FUNCTION_BLOCK ILOCK_2_E_AX (* Event-driven bistable and Toggle with Dual Interlock (Adapter) *)
  (* Standard: 61499-1 Annex A; Description: Copyright (c) 2017, 2024 fortiss GmbH, HR Agrartechnik GmbH This program and the accompanying materials are made available under the terms of the Eclipse Public License 2.0 which is available at https://www.eclipse.org/legal/epl-2.0/ SPDX-License-Identifier: EPL-2.0 *)
  (* Version 3.0, 2025-04-14, Patrick Aigner, changed package *)
  (* Version 1.1, 2024-08-27, Franz Höpfinger, HR Agrartechnik GmbH, Copy E_SR and make this FB *)
  (* Version 1.0, 2017-09-22, Alois Zoitl, fortiss GmbH, initial API and implementation and/or initial documentation *)
  PACKAGE logiBUS::signalprocessing::interlock;
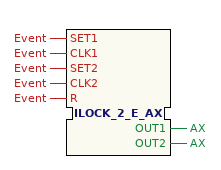
  EVENT_INPUT
    SET1; (* Set output OUT1 *)
    CLK1; (* Clock for triggering a output toggle on OUT1 *)
    SET2; (* Set output OUT2 *)
    CLK2; (* Clock for triggering a output toggle on OUT2 *)
    R; (* Reset all outputs *)
  END_EVENT
  PLUGS
    OUT1 : adapter::types::unidirectional::AX; (* value of flip flop *)
    OUT2 : adapter::types::unidirectional::AX; (* value of flip flop *)
  END_PLUGS
  VAR
    EDGE1 : BOOL := FALSE;
    EDGE2 : BOOL := FALSE;
  END_VAR
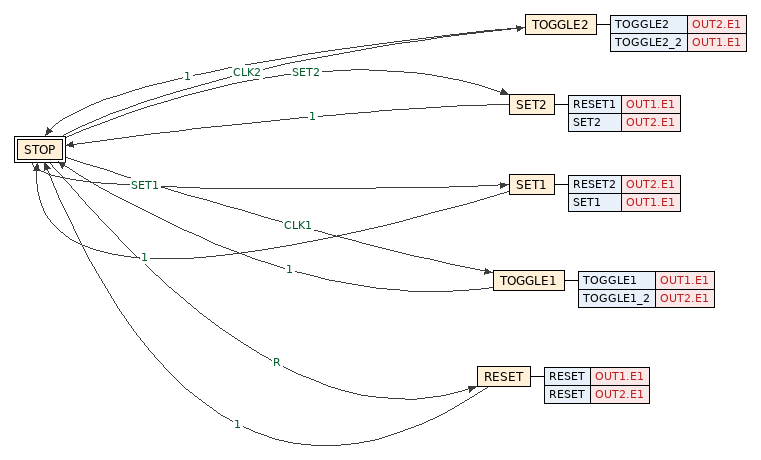
  EC_STATES
    STOP; (* Initial State *)
    TOGGLE1 : TOGGLE1 -> OUT1.E1, TOGGLE1_2 -> OUT2.E1;
    RESET : RESET -> OUT1.E1, RESET -> OUT2.E1;
    SET1 : RESET2 -> OUT2.E1, SET1 -> OUT1.E1;
    SET2 : RESET1 -> OUT1.E1, SET2 -> OUT2.E1;
    TOGGLE2 : TOGGLE2 -> OUT2.E1, TOGGLE2_2 -> OUT1.E1;
  END_STATES
  EC_TRANSITIONS
    STOP TO SET1 := SET1;
    STOP TO SET2 := SET2;
    STOP TO TOGGLE1 := CLK1;
    STOP TO TOGGLE2 := CLK2;
    STOP TO RESET := R;
    TOGGLE1 TO STOP := 1;
    SET1 TO STOP := 1;
    SET2 TO STOP := 1;
    TOGGLE2 TO STOP := 1;
    RESET TO STOP := 1;
  END_TRANSITIONS
  ALGORITHM SET1 IN ST:
OUT1.D1 := TRUE;
OUT2.D1 := FALSE;
EDGE1 := FALSE;
EDGE2 := FALSE;
  END_ALGORITHM
  ALGORITHM SET2 IN ST:
OUT1.D1 := FALSE;
OUT2.D1 := TRUE;
EDGE1 := FALSE;
EDGE2 := FALSE;
  END_ALGORITHM
  ALGORITHM TOGGLE1 IN ST:
IF NOT EDGE1 THEN
	OUT1.D1 := NOT OUT1.D1;
END_IF;
EDGE1 := TRUE;
EDGE2 := FALSE;
  END_ALGORITHM
  ALGORITHM TOGGLE1_2 IN ST:
OUT2.D1 := FALSE;
  END_ALGORITHM
  ALGORITHM TOGGLE2 IN ST:
IF NOT EDGE2 THEN
	OUT2.D1 := NOT OUT2.D1;
END_IF;
EDGE1 := FALSE;
EDGE2 := TRUE;
  END_ALGORITHM
  ALGORITHM TOGGLE2_2 IN ST:
OUT1.D1 := FALSE;
  END_ALGORITHM
  ALGORITHM RESET IN ST:
OUT1.D1 := FALSE;
OUT2.D1 := FALSE;
EDGE1 := FALSE;
EDGE2 := FALSE;
  END_ALGORITHM
  ALGORITHM RESET1 IN ST:
OUT1.D1 := FALSE;
EDGE1 := FALSE;
EDGE2 := FALSE;
  END_ALGORITHM
  ALGORITHM RESET2 IN ST:
OUT2.D1 := FALSE;
EDGE1 := FALSE;
EDGE2 := FALSE;
  END_ALGORITHM
END_FUNCTION_BLOCK
